Universal Robots URScript: dus5_probe_l.script

# =============================================================================
#  dus5_probe_l.script — dusan_v5
#  호의 양 끝점을 반지름·호각으로 **먼저 계산**하고, 원점(이 중 Y- 끝)은
#  그 계산값으로 접근해 실제 벽 접촉으로 다시 보정한다.
#
#  펜던트에서 "4_probe_left" 자리에 스크립트 노드를 파일(File) 모드로 넣고 지정한다.
#
#  ※ def main() 으로 감싸지 말 것 (펜던트가 호출하지 않는다)
#  ※ 최상위에 global 을 쓰지 말 것 (preamble 이 이미 선언·대입해 뒀다)
#  ※ if / while 은 반드시 end 로 닫을 것
#
#  센서가 중앙 하나뿐이라 계산만으로 끝내면, 도면 반지름이 실제 벽과 조금만
#  달라도(또는 벽이 완전한 원통이 아니어도) 원점이 벽에서 뜨거나 파고든다.
#  그래서 계산값은 "여기쯤일 것이다"라는 접근 목표로만 쓰고, 그 자리에 가서
#  중앙과 똑같이 눌림 센서로 다시 찾는다 — probe_c 의 pc_press() 와 같은
#  방식이다. Y- 끝(p_r_pose)은 여기서는 계산만 해 두고, dus5_probe_r.script가
#  같은 방식으로 실측한다.
#
#  기하: 중앙 접점 P 에서 TCP +Z 로 R 만큼 간 곳이 곡률 중심 O 다
#  (바깥 볼록면을 훑으므로 중심은 벽 뒤에 있다). O 를 베이스 Z 로 t 만큼 돌린 뒤
#  다시 로컬 -Z 로 R 만큼 나오면 호 위의 점이 되고, **손 방향도 그 점의
#  법선으로 같이 돌아간다** — servoj 호에 그대로 쓸 수 있는 자세다.
# =============================================================================

def al_w1(a, v):
  if (v > 32000):
    v = 32000
  end
  if (v < -32000):
    v = -32000
  end
  write_port_register(a, floor(v + 0.5))
end


def al_w6(a, p):
  al_w1(a, p[0] * 10000)
  al_w1(a + 1, p[1] * 10000)
  al_w1(a + 2, p[2] * 10000)
  al_w1(a + 3, p[3] * 1000)
  al_w1(a + 4, p[4] * 1000)
  al_w1(a + 5, p[5] * 1000)
end


def al_arc(mid, th):
  # 중앙 접점 mid 에서 호를 따라 th [rad] 만큼 돌아간 점(자세 포함).
  #
  # 원통은 세워져 있으므로 호는 **수평면** 안에 있다. 그래서
  #   (1) 곡률 중심 O 는 접점에서 '전진 방향(TCP +Z)의 **수평 성분**'으로 R.
  #       TCP +Z 가 조금 기울어 있어도 수평 성분만 써야 반지름이 맞는다.
  #   (2) 회전은 O 를 지나는 **수직축(베이스 Z)** 으로 한다.
  #       툴 로컬 Z 로 돌리면 호가 수평면을 벗어나 현이 짧아진다.
  # 자세도 같이 돌아가므로 각 점에서 손이 그 자리의 법선을 본다.
  if (scan_radius <= 0):
    return mid
  end
  fwd = pose_trans(mid, [0, 0, 1.0, 0, 0, 0])
  dx = fwd[0] - mid[0]
  dy = fwd[1] - mid[1]
  n = sqrt(dx * dx + dy * dy)
  if (n < 0.0001):
    # 전진 방향이 거의 수직이다 = 벽을 보고 있지 않다. 그대로 둔다.
    return mid
  end
  r = scan_radius * 0.001
  # 곡률 중심은 **프로브 중심**(툴 플랜지 + EOAT 오프셋 eoat_ofs)에서 R 이다.
  # 플랜지에서 잡으면 오프셋 z 만큼 중심이 어긋나, 벽 위로 훑는 호가 L*(R-z)/R 로
  # 짧아지고 양 끝이 벽을 파고든다. 플랜지 pose 를 이 중심으로 돌리면 프로브
  # 중심도 같이 돌아 벽(반지름 R) 위에 그대로 남는다.
  tip = pose_trans(mid, eoat_ofs)
  o_t = [tip[0] + dx / n * r, tip[1] + dy / n * r, 0, 0, 0, 0]
  return pose_trans(o_t, pose_trans([0, 0, 0, 0, 0, th],
                   pose_trans(pose_inv(o_t), mid)))
end


def al_push():
  # 센서가 적정 눌림을 잡은 자리에서 push_offset [mm] 만큼 **더 민다**(TCP +Z).
  # 0 이면 아무것도 안 한다. 벽을 누르는 중이라 천천히(v_l / 10) 민다.
  # 이 뒤에 잡는 접점 pose 가 곧 스캔 경로가 되므로, 스캔 전체가 이만큼
  # 더 눌린 채로 돈다.
  if (push_offset > 0):
    movel(pose_trans(get_actual_tcp_pose(), [0, 0, push_offset * 0.001, 0, 0, 0]),
       a = a_l, v = v_l / 10.0)
  end
end


def al_step(dmm):
  # TCP 기준 Z 로 dmm [mm] 만큼 움직인다. 음수가 전진(벽 쪽) — dmm 부호의
  # 의미는 예전(Y축) 그대로 두고, 축만 Y에서 Z로 바꾼다(그래서 부호가
  # 한 번 뒤집힌다: 예전 [0,dmm,0,0,0,0] -> 이제 [0,0,-dmm,0,0,0]).
  movel(pose_trans(get_actual_tcp_pose(), [0, 0, -dmm * 0.001, 0, 0, 0]),
     a = a_l, v = v_l / 3.0)
end


def al_rush(t):
  movel(t, a = a_l, v = v_l / 3.0)
end


def al_press(target):
  # target 자세(계산값) 그대로, 그 지점의 로컬 +Z 로 전진해 실제 벽
  # 접촉을 찾는다 — probe_c 의 pc_press() 와 같은 방식이다.
  # 반환: 실제로 닿은 pose(자세는 target 유지, 위치만 실측으로 보정됨).
  # 못 찾으면 계산값으로 조용히 넘어가지 않는다 — 아래에서 멈춘다.
  global n_hit
  far = pose_trans(target, [0, 0, seek_limit * 0.001, 0, 0, 0])
  mv_h = start_thread(al_rush, (far,), detach_mode = False)
  while (True):
    if (get_standard_digital_in(di_touch) or get_standard_digital_in(di_limit)):
      stop_thread(mv_h)
      stopl(1.2)
      break
    end
    if (pose_dist(get_actual_tcp_pose(), far) < 0.0005):
      stop_thread(mv_h)
      stopl(1.2)
      break
    end
    sync()
  end

  tries = 0
  while (get_standard_digital_in(di_limit) and tries < seek_tries):
    tries = tries + 1
    al_step(seek_step)
    sync()
  end

  tries = 0
  while (get_standard_digital_in(di_touch) == False and tries < seek_tries):
    tries = tries + 1
    al_step(-seek_step)
    sync()
  end

  if (get_standard_digital_in(di_touch)):
    n_hit = n_hit + 1
    al_push()
    return get_actual_tcp_pose()
  end
  # 계산값 대신 쓸 값이 없다 — 원점이 실측 없이 계산값으로 넘어가면
  # 스캔 전체가 잘못된 좌표로 돌게 되므로, 실패는 반드시 멈춰서 알려야 한다.
  popup(s = "PROBE_L: WALL CONTACT NOT FOUND", title = "dusan_v5", blocking = True)
  write_port_register(299, 2)
  write_port_register(290, 9)
  halt()
  return target
end


write_port_register(290, 3)

# 양 끝을 다 계산해 놓고, 베이스 Y 가 작은 쪽을 Y-(원점), 큰 쪽을 Y+ 로 나눈다.
# 손이 어느 방향을 보고 있느냐에 따라 +t 가 어느 쪽으로 갈지 달라지므로
# 부호를 미리 못 박지 않고 실제 좌표로 가른다.
# 호가 0 이면(반지름 0 또는 arc_run 0) al_arc 가 중앙점을 그대로 돌려줘
# 양 끝이 중앙과 겹친다. 그 상태로 진행하면 나중에 dus5_pass_r 의 servoj 호가
# "Target pose ... coincident with auxiliary pose" 로 죽는데, 그 문구만
# 보고는 원인을 알 수 없다. 여기서 값을 짚어 멈춘다.
if (scan_radius <= 0 or arc_half == 0):
  popup(s = "ARC IS ZERO: check radius(260) and arc length(256)",
        title = "dusan_v5", blocking = True)
  write_port_register(299, 4)
  write_port_register(290, 9)
  halt()
end

end_a = al_arc(p_c_pose, arc_half)
end_b = al_arc(p_c_pose, -arc_half)
# 반시계 방향으로 훑는다. 원점은 베이스 Y 가 **큰** 쪽 끝이고, 거기서
# Y 가 줄어드는 방향으로 한 줄을 지난다. (예전에는 반대였다 — Y 가 작은
# 쪽이 원점이었다.) 발행하는 좌표는 dus5_init 의 pub_rel 이 Rz 180 도로
# 뒤집어 내보내므로, 이렇게 훑어도 Y 는 계속 + 로만 커진다.
if (end_a[1] >= end_b[1]):
  zero_est = end_a
  p_r_pose = end_b
else:
  zero_est = end_b
  p_r_pose = end_a
end

# 계산한 원점(zero_est)의 대기 지점(TCP -Z 로 물러난 곳)까지 안전하게
# 이동한 뒤, 그 자세 그대로 전진해 실제 벽 접촉으로 원점을 보정한다.
#
# 여기 오기 전 위치(중앙, p_c_pose)에서 l_stand 까지는 호의 절반 가까이
# 자세가 크게 돌아간다. 한때 movej(get_inverse_kin(...))로 바꿨었는데,
# 좌우 이동은 movel(직선)로 가도록 되돌린다.
l_stand = pose_trans(zero_est, [0, 0, -probe_dist * 0.001, 0, 0, 0])
movel(l_stand, a = a_l, v = v_l)
zero_pose = al_press(zero_est)

# 이 자리가 원점이자 호의 시작점이다 (회전값 포함).
p_lx = zero_pose[0]
write_port_register(301, floor(p_lx * 10000 + 0.5))
al_w6(350, zero_pose)
zero_inv = pose_inv(zero_pose)
zero_ok = True

# ---- 호 위 위치를 실시간으로 내보내기 위한 기준 ---------------------------
# TPAC 은 스캔 축 위치로 **호 길이**를 받아야 한다. 좌표를 그대로 주면
# 현(1031.8)으로 7% 눌리고, 게다가 호 위치에 비례하지 않아 1/4·3/4 지점에서
# 14.6mm 씩 어긋난다(C-scan 이 앞뒤로 밀려 찍힌다).
# 곡률 중심과 원점의 방위각을 남겨 두면, 발행 스레드가 매 주기
#   s = R * |현재각 - 원점각|
# 으로 호 위 실제 거리를 계산할 수 있다.
if (scan_radius > 0):
  fwd0 = pose_trans(p_c_pose, [0, 0, 1.0, 0, 0, 0])
  d0x = fwd0[0] - p_c_pose[0]
  d0y = fwd0[1] - p_c_pose[1]
  n0 = sqrt(d0x * d0x + d0y * d0y)
  if (n0 > 0.0001):
    # 곡률 중심·원점 방위각도 프로브 중심 기준(eoat_ofs) — 호 계산과 같은 점이어야
    # 286/287 의 호 위 거리가 벽 위 실제 호 길이와 같다.
    c_tip = pose_trans(p_c_pose, eoat_ofs)
    z_tip = pose_trans(zero_pose, eoat_ofs)
    arc_ox = c_tip[0] + d0x / n0 * scan_radius * 0.001
    arc_oy = c_tip[1] + d0y / n0 * scan_radius * 0.001
    arc_phi0 = atan2(z_tip[1] - arc_oy, z_tip[0] - arc_ox)
    arc_ok = True
  end
end

n_probe = n_probe + 1
write_port_register(304, n_probe)
write_port_register(305, n_hit)

# 벽에서 물러난다 (다음 동작에서 곡면을 가로지르지 않도록) — 좌우 이동은
# movel(직선)로 간다.
movel(l_stand, a = a_l, v = v_l)
